TEXTLIST TL_E_MESSAGETYPE
  0 = 'eMessageEmpty'
  1 = 'eMessageError'
  2 = 'eMessageWarning'
  3 = 'eMessageInfo'
  4 = 'eMessageVerbose'
   = ''
END_TEXTLIST

(* stored: Version 1.1.0.1
   TextList TL_E_MESSAGETYPE: Id {aab85940-c774-4fa2-9a99-58d135e39408} *)
